{attribute 'GeneratedUsingTerminal: EK1122-0000-0018'}
{attribute addProperty BoxType "EK1122-0000-0018"}
{attribute addProperty Id "Beckhoff_ER7xxxsub_EK1100EK1100_AB5A94672A_0001_ER7041_0002_0024ER7041_5461F6FA53A_0002_ER7041_0002_0025ER7041_5461F6FA53A_0003_ER7041_1002_0024ER7041_5461F6FA53A_0004_ER7041_1002_0025ER7041_5461F6FA53A_0005_ER7041_2002_0024ER7041_5461F6FA53A_0006_ER7041_2002_0025ER7041_5461F6FA53A_0007_ER7041_3002_0021ER7041_583AD35554A_0008_ER7041_3002_0022ER7041_583AD35554A_0009_ER7342_0002_0020ER7342_2F848FE386A_0010_ER7342_0002_0021ER7342_2F848FE386A_0011_ER7342_0002_0022ER7342_2F848FE386"}
{attribute addProperty CRC "3492048949"}
{attribute addProperty Size "686"}
TYPE Beckhoff_ER7xxxEK1122_D0247035 EXTENDS EK1122_AB5A9467 :
STRUCT
	{attribute addProperty Name "Beckhoff_ER7xxxsub_EK1100"}
	{attribute addProperty PreviousPort "Beckhoff ER7xxxEK1122 : D"}
	Beckhoff_ER7xxxsub_EK1100 : EK1100_AB5A9467;
	{attribute addProperty Name "A_0001_ER7041_0002_0024"}
	{attribute addProperty PreviousPort "Beckhoff ER7xxxsub EK1100 : C"}
	A_0001_ER7041_0002_0024 : ER7041_5461F6FA;
	{attribute addProperty Name "A_0002_ER7041_0002_0025"}
	{attribute addProperty PreviousPort "A_0001(ER7041-0002-0024) : B"}
	A_0002_ER7041_0002_0025 : ER7041_5461F6FA;
	{attribute addProperty Name "A_0003_ER7041_1002_0024"}
	{attribute addProperty PreviousPort "A_0002(ER7041-0002-0025) : B"}
	A_0003_ER7041_1002_0024 : ER7041_5461F6FA;
	{attribute addProperty Name "A_0004_ER7041_1002_0025"}
	{attribute addProperty PreviousPort "A_0003(ER7041-1002-0024) : B"}
	A_0004_ER7041_1002_0025 : ER7041_5461F6FA;
	{attribute addProperty Name "A_0005_ER7041_2002_0024"}
	{attribute addProperty PreviousPort "A_0004(ER7041-1002-0025) : B"}
	A_0005_ER7041_2002_0024 : ER7041_5461F6FA;
	{attribute addProperty Name "A_0006_ER7041_2002_0025"}
	{attribute addProperty PreviousPort "A_0005(ER7041-2002-0024) : B"}
	A_0006_ER7041_2002_0025 : ER7041_5461F6FA;
	{attribute addProperty Name "A_0007_ER7041_3002_0021"}
	{attribute addProperty PreviousPort "A_0006(ER7041-2002-0025) : B"}
	A_0007_ER7041_3002_0021 : ER7041_583AD355;
	{attribute addProperty Name "A_0008_ER7041_3002_0022"}
	{attribute addProperty PreviousPort "A_0007(ER7041-3002-0021) : B"}
	A_0008_ER7041_3002_0022 : ER7041_583AD355;
	{attribute addProperty Name "A_0009_ER7342_0002_0020"}
	{attribute addProperty PreviousPort "A_0008(ER7041-3002-0022) : B"}
	A_0009_ER7342_0002_0020 : ER7342_2F848FE3;
	{attribute addProperty Name "A_0010_ER7342_0002_0021"}
	{attribute addProperty PreviousPort "A_0009(ER7342-0002-0020) : B"}
	A_0010_ER7342_0002_0021 : ER7342_2F848FE3;
	{attribute addProperty Name "A_0011_ER7342_0002_0022"}
	{attribute addProperty PreviousPort "A_0010(ER7342-0002-0021) : B"}
	A_0011_ER7342_0002_0022 : ER7342_2F848FE3;
END_STRUCT
END_TYPE

(* stored: Version 1.2.0.0, ProductVersion 3.1.4024.9
   DUT Beckhoff_ER7xxxEK1122_D0247035: Id {ca4a2232-407e-44db-8cd5-b37a036b45d8} *)
